(* IEC 61131-3 sources: generating_plc_code_with_llms/Code#1/ChatGPT_4/second run, 21 files *)

(* ---- 14.st ---- *)
// 60.33s
// 2
FUNCTION FC1001 : BOOL
VAR_INPUT
    measuredValue : REAL;  // Sensor reading
    switchingValue : REAL; // Predetermined switching value
    hysteresis : REAL;     // Hysteresis in percentage of the switching value
END_VAR

VAR
    hysteresisValue : REAL;
    static lastState : BOOL := FALSE;
END_VAR

// Calculate the hysteresis value
hysteresisValue := switchingValue * (hysteresis / 100.0);

// Switching logic with hysteresis
IF measuredValue > (switchingValue + hysteresisValue) THEN
    lastState := TRUE;  // Turn on the output
ELSIF measuredValue < (switchingValue - hysteresisValue) THEN
    lastState := FALSE; // Turn off the output
END_IF

FC1001 := lastState;

END_FUNCTION

(* ---- 15.st ---- *)
// 48.69s
// 2
FUNCTION FC1002 : BOOL
VAR_INPUT
    sensorDetected : BOOL; // TRUE if ultrasonic sensor detects something
    switchEA : BOOL;       // TRUE if the monitoring system is switched on
END_VAR

VAR_OUTPUT
    hornPHU : BOOL;        // Horn for acoustic warning signal
    alarmPAL : BOOL;       // Alarm signal
    indicatorP1 : BOOL;    // Indicator for monitoring system status
END_VAR

VAR
    detectionStartTime : TIME;
    systemActive : BOOL;
    static lastDetectionTime : TIME := 0;
END_VAR

// System control logic
IF switchEA THEN
    indicatorP1 := TRUE;  // Monitoring system is active
    systemActive := TRUE;

    IF sensorDetected THEN
        IF NOT hornPHU THEN
            detectionStartTime := TIME();  // Start the detection timer
        END_IF

        hornPHU := TRUE;  // Activate horn

        // Check if detection lasts longer than 3 seconds
        IF TIME() - detectionStartTime > T#3s THEN
            hornPHU := FALSE;   // Turn off horn
            alarmPAL := TRUE;   // Activate alarm
        END_IF
    ELSE
        hornPHU := FALSE;
        alarmPAL := FALSE;
        detectionStartTime := 0;
    END_IF
ELSE
    // Reset all outputs and states when the system is switched off
    hornPHU := FALSE;
    alarmPAL := FALSE;
    indicatorP1 := FALSE;
    systemActive := FALSE;
    detectionStartTime := 0;
END_IF

FC1002 := systemActive;

END_FUNCTION

(* ---- 18.st ---- *)
// 34.21s
// 4
FUNCTION FC1003 : REAL
VAR_INPUT
    digitalValue : REAL;   // Digital input value (e.g., 0 to 255)
    IN_MIN : REAL;         // Lower limit of the input range
    IN_MAX : REAL;         // Upper limit of the input range
    OUT_MIN : REAL;        // Lower limit of the output range (e.g., -20°C)
    OUT_MAX : REAL;        // Upper limit of the output range (e.g., 40°C)
END_VAR

VAR
    scaleFactor : REAL;
    offset : REAL;
END_VAR

BEGIN
    // Calculate the scale factor and offset for linear mapping
    scaleFactor := (OUT_MAX - OUT_MIN) / (IN_MAX - IN_MIN);
    offset := OUT_MIN - scaleFactor * IN_MIN;

    // Apply linear mapping
    FC1003 := scaleFactor * digitalValue + offset;
END_FUNCTION

(* ---- 19.st ---- *)
// 39.94s
// 2
FUNCTION_BLOCK FB1005
VAR_INPUT
    Laser1 : REAL;      // Measurement from Laser 1
    Laser2 : REAL;      // Measurement from Laser 2
    S1 : BOOL;          // Sensor to start/end measurement
    V_MAX : REAL;       // Upper tolerance limit
    V_MIN : REAL;       // Lower tolerance limit
END_VAR

VAR_OUTPUT
    M_MAX : REAL;       // Maximum measured thickness
    M_MIN : REAL;       // Minimum measured thickness
    P1 : BOOL;          // Reject indicator
END_VAR

VAR
    measuring : BOOL := FALSE;  // Indicates if currently measuring
    currentThickness : REAL;
END_VAR

BEGIN
    IF S1 THEN
        IF NOT measuring THEN
            // Start of a new measurement
            M_MAX := -REAL_MAX;
            M_MIN := REAL_MAX;
            measuring := TRUE;
            P1 := FALSE;
        END_IF

        // Calculate current thickness
        currentThickness := ABS(Laser1 - Laser2);

        // Update M_MAX and M_MIN
        IF currentThickness > M_MAX THEN
            M_MAX := currentThickness;
        END_IF

        IF currentThickness < M_MIN THEN
            M_MIN := currentThickness;
        END_IF

        // Check if the current measurement is out of tolerance
        IF (M_MAX > V_MAX) OR (M_MIN < V_MIN) THEN
            P1 := TRUE;  // Plate is scrap
        END_IF
    ELSE
        IF measuring THEN
            // End of measurement
            measuring := FALSE;
        END_IF
    END_IF
END_FUNCTION_BLOCK

(* ---- 21.st ---- *)
// 119.91s
// 3
FUNCTION_BLOCK BURNER
VAR_INPUT
    IN : BOOL;                // Start signal
    OVER_TEMP : BOOL;         // Boiler over-temperature signal
    OIL_TEMP : BOOL;          // Oil temperature readiness signal
    STAGE2 : BOOL;            // Signal to start stage 2
    RST : BOOL;               // Reset signal
END_VAR

VAR_OUTPUT
    PRE_HEAT : BOOL;          // Pre-heating signal
    MOTOR : BOOL;             // Motor operation signal
    IGNITION : BOOL;          // Ignition signal
    OIL_VALVE : BOOL;         // Oil valve open signal
    FAIL : BOOL;              // Failure signal
    STATUS : INT;             // Status code output
END_VAR

VAR
    TIMER : TON;              // Timer for managing delays
    currentStage : INT := 0;  // Current operation stage
    lockoutTimer : TON;       // Timer for managing lockout period
END_VAR

// Constants for timing (to be adjusted as per requirements)
VAR CONSTANT
    PRE_HEAT_TIME : TIME := T#30s;
    PRE_VENTILATION_TIME : TIME := T#15s;
    PRE_IGNITE_TIME : TIME := T#5s;
    SAFETY_TIME : TIME := T#10s;
    POST_IGNITE_TIME : TIME := T#5s;
    STAGE2_DELAY : TIME := T#60s;
    LOCKOUT_TIME : TIME := T#300s;
    MULTIPLE_IGNITION : BOOL := TRUE;  // Can be set based on requirements
END_VAR

// State machine logic
IF OVER_TEMP THEN
    // Immediate stop and report error 9
    STATUS := 9;
    FAIL := TRUE;
    ResetOutputs();
ELSIF RST AND NOT lockoutTimer.Q THEN
    // Resetting the burner
    FAIL := FALSE;
    STATUS := 110; // Standby
    currentStage := 0;
    ResetOutputs();
ELSIF IN THEN
    CASE currentStage OF
    0:  // Start sequence
        PRE_HEAT := TRUE;
        TIMER(IN := TRUE, PT := PRE_HEAT_TIME);
        IF OIL_TEMP THEN
            currentStage := 1;
            PRE_HEAT := FALSE;
            MOTOR := TRUE;
        ELSIF TIMER.Q THEN
            // Pre-heat failure
            FAIL := TRUE;
            STATUS := 1;
            currentStage := -1;  // Move to error state
        END_IF;
    1:  // Motor and ventilation
        TIMER(IN := TRUE, PT := PRE_VENTILATION_TIME);
        IF TIMER.Q THEN
            currentStage := 2;
            MOTOR := FALSE;  // Assuming motor should stop before ignition, adjust as needed
            IGNITION := TRUE;
        END_IF;
    2:  // Ignition and oil valve
        TIMER(IN := TRUE, PT := PRE_IGNITE_TIME);
        IF TIMER.Q THEN
            OIL_VALVE := TRUE;
            TIMER(IN := TRUE, PT := SAFETY_TIME);  // Start safety timer
            currentStage := 3;
        END_IF;
    3:  // Safety check
        IF NOT TIMER.Q THEN
            // Assume flame detected, proceed
            STATUS := 112;  // Burner running on stage 1
            currentStage := 4;
        ELSE
            // Safety time passed without flame
            FAIL := TRUE;
            STATUS := 4;
            currentStage := -1;  // Move to error state
        END_IF;
    4:  // Stage 2 check
        IF STAGE2 THEN
            TIMER(IN := TRUE, PT := STAGE2_DELAY);
            IF TIMER.Q THEN
                STATUS := 113;  // Burner running at stage 2
                // Implement stage 2 functionality as required
            END_IF;
        END_IF;
    -1: // Error state
        ResetOutputs();
        lockoutTimer(IN := TRUE, PT := LOCKOUT_TIME);  // Start lockout timer
        IF lockoutTimer.Q THEN
            // Lockout period finished, ready for reset
            currentStage := 0;
            FAIL := FALSE;
            STATUS := 110; // Back to standby after reset
        END_IF;
    END_CASE;
END_IF;

// Helper procedure to reset outputs
PROCEDURE ResetOutputs();
BEGIN
    PRE_HEAT := FALSE;
    MOTOR := FALSE;
    IGNITION := FALSE;
    OIL_VALVE := FALSE;
    TIMER(IN := FALSE, PT := T#0s);  // Reset timer
END_PROCEDURE

END_FUNCTION_BLOCK

(* ---- 1.st ---- *)
//16.57s
//4
PROGRAM AlarmControl
VAR
    xAlarm1: BOOL; // Alarm 1
    xAlarm2: BOOL; // Alarm 2
    xAllOn: BOOL;  // Signal to set all alarms
    xAllOff: BOOL; // Signal to reset all alarms
END_VAR

// When the xAllOn signal is active, set both alarms to TRUE
IF xAllOn THEN
    xAlarm1 := TRUE;
    xAlarm2 := TRUE;
    // Reset the signals after processing
    xAllOn := FALSE;
END_IF

// When the xAllOff signal is active, set both alarms to FALSE
IF xAllOff THEN
    xAlarm1 := FALSE;
    xAlarm2 := FALSE;
    // Reset the signals after processing
    xAllOff := FALSE;
END_IF

END_PROGRAM

(* ---- 10.st ---- *)
//16.26s
//4
PROGRAM SigmoidFunction
VAR
    x: REAL;        // Input for the sigmoid function
    sigmoid: REAL;  // Result of the sigmoid function
END_VAR

// Calculate the sigmoid function
sigmoid := 1 / (1 + EXP(-x));

END_PROGRAM

(* ---- 11.st ---- *)
//19.66s
//4
PROGRAM SignFunction
VAR
    x: REAL;        // Input variable
    signum: INT;    // Output variable (-1, 0, 1)
END_VAR

// Calculate the signum of the variable x
IF x < 0 THEN
    signum := -1;
ELSIF x > 0 THEN
    signum := 1;
ELSE
    signum := 0;
END_IF;

END_PROGRAM

(* ---- 12.st ---- *)
//14.62s
//4
PROGRAM HyperbolicSine
VAR
    x: REAL;           // Input variable
    sinh_x: REAL;      // Result of hyperbolic sine of x
END_VAR

// Calculate the hyperbolic sine of x
sinh_x := (EXP(x) - EXP(-x)) / 2;

END_PROGRAM

(* ---- 13.st ---- *)
//30.69s
//2
PROGRAM SearchNumber
VAR
    RandomNumbers: ARRAY[1..100] OF INT; // Array containing 100 random numbers
    Found: BOOL; // TRUE if the number 10 is found, FALSE otherwise
    i: INT; // Index used for iterating through the list
END_VAR

i := 1; // Initialize index
Found := FALSE; // Initialize Found as FALSE

REPEAT
    IF RandomNumbers[i] = 10 THEN
        Found := TRUE; // Set Found to TRUE if number 10 is found
        EXIT; // Exit the loop if number 10 is found
    END_IF;
    i := i + 1; // Increment index
UNTIL i > 100; // Continue until the end of the list is reached

IF Found THEN
    // Number 10 was found in the list
    // Additional actions can be taken here if necessary
ELSE
    // Number 10 was not found in the list
    // Additional actions can be taken here if necessary
END_IF;

END_PROGRAM

(* ---- 16.st ---- *)
//41.0s
//4
PROGRAM TrafficLightControl
VAR
    North_green, North_yellow, North_red: BOOL; // North traffic lights
    East_green, East_yellow, East_red: BOOL; // East traffic lights
    CycleTimer: TON; // Timer for controlling the cycle
END_VAR

// Start the cycle timer
CycleTimer(IN:=TRUE, PT:=T#10000ms);

// Control North traffic light
IF CycleTimer.ET < T#5000ms THEN
    // Between 0ms and 5000ms, North is green and East is red
    North_green := TRUE;
    North_yellow := FALSE;
    North_red := FALSE;

    East_green := FALSE;
    East_yellow := FALSE;
    East_red := TRUE;
ELSIF CycleTimer.ET < T#5500ms THEN
    // Between 5000ms and 5500ms, North turns yellow
    North_green := FALSE;
    North_yellow := TRUE;
    North_red := FALSE;

    East_green := FALSE;
    East_yellow := FALSE;
    East_red := TRUE;
ELSE
    // After 5500ms, North is red
    North_green := FALSE;
    North_yellow := FALSE;
    North_red := TRUE;
END_IF;

// Control East traffic light
IF CycleTimer.ET >= T#5500ms AND CycleTimer.ET < T#9500ms THEN
    // Between 5500ms and 9500ms, East is green
    East_green := TRUE;
    East_yellow := FALSE;
    East_red := FALSE;
ELSIF CycleTimer.ET >= T#9500ms THEN
    // Between 9500ms and 10000ms, East turns yellow
    East_green := FALSE;
    East_yellow := TRUE;
    East_red := FALSE;
END_IF;

// Reset the timer after the cycle completes
IF CycleTimer.ET >= CycleTimer.PT THEN
    CycleTimer.IN := FALSE; // Stop the timer
    CycleTimer( IN:=FALSE ); // Reset the timer
    CycleTimer.IN := TRUE; // Restart the timer for the next cycle
END_IF;

END_PROGRAM

(* ---- 17.st ---- *)
//39.92s
//2
PROGRAM WeatherStation
VAR
    aiTemperature: INT; // Analog input value for temperature
    aiHumidity: INT; // Analog input value for humidity
    rTemperatureC: REAL; // Scaled temperature in degrees Celsius
    rHumidityPct: REAL; // Scaled humidity in percent
    DisplayText: STRING; // Text to be displayed
END_VAR

// Assuming aiTemperature and aiHumidity are scaled appropriately to 0-100% for the 0-32767 range
rTemperatureC := (REAL(aiTemperature) / 32767) * 100; // Convert to degrees Celsius (example scaling)
rHumidityPct := (REAL(aiHumidity) / 32767) * 100; // Convert to percent (example scaling)

IF rTemperatureC < 18 THEN
    DisplayText := 'Cold';
ELSIF rTemperatureC > 25 THEN
    DisplayText := 'Hot';
ELSE
    // Temperature is between 18 and 25 degrees Celsius, check humidity
    IF rHumidityPct >= 40 AND rHumidityPct <= 75 THEN
        DisplayText := 'Opt'; // Optimum conditions
    ELSE
        DisplayText := 'Temp. OK'; // Temperature is okay, but humidity is not in the optimum range
    END_IF;
END_IF;

END_PROGRAM

(* ---- 2.st ---- *)
//18.14s
//4
FUNCTION Factorial: LINT
VAR_INPUT
    n: INT; // Input value to calculate the factorial of
END_VAR
VAR
    i: INT;
    result: LINT := 1; // Initialize result to 1 (0! = 1)
END_VAR

FOR i := 1 TO n DO
    result := result * i;
END_FOR

Factorial := result; // Return the factorial result
END_FUNCTION

PROGRAM BinomialCoefficient
VAR
    n: INT; // Total number of items
    k: INT; // Number of items to choose
    binomCoeff: LINT; // Binomial coefficient result
END_VAR

// Ensure that 0 <= k <= n, otherwise the binomial coefficient is not defined
IF k >= 0 AND k <= n THEN
    binomCoeff := Factorial(n) / (Factorial(k) * Factorial(n - k));
ELSE
    binomCoeff := 0; // If the condition is not met, the result is 0
END_IF

END_PROGRAM

(* ---- 20.st ---- *)
// 48.24s
// 4
PROGRAM InterlockProgram
VAR
    I1, I2 : BOOL;       // Inputs
    Q1, Q2 : BOOL;       // Outputs
    TL : TIME;           // Dead time between outputs
    LastQ1Time, LastQ2Time : TIME;  // Time trackers for Q1 and Q2
END_VAR

BEGIN
    // Update time trackers
    IF Q1 THEN
        LastQ1Time := TIME();
    END_IF
    IF Q2 THEN
        LastQ2Time := TIME();
    END_IF

    // Logic for Q1
    IF I1 AND NOT Q2 AND (TIME() - LastQ2Time > TL) THEN
        Q1 := TRUE;
    ELSE
        Q1 := FALSE;
    END_IF

    // Logic for Q2
    IF I2 AND NOT Q1 AND (TIME() - LastQ1Time > TL) THEN
        Q2 := TRUE;
    ELSE
        Q2 := FALSE;
    END_IF
END_PROGRAM

(* ---- 3.st ---- *)
//24.56s
//2
FUNCTION Fibonacci: LINT
VAR_INPUT
    n: INT; // The n-th Fibonacci number to calculate
END_VAR
VAR
    a: LINT := 0; // First number in the sequence
    b: LINT := 1; // Second number in the sequence
    i: INT;
    temp: LINT;
END_VAR

IF n = 0 THEN
    RETURN 0; // The 0th Fibonacci number is 0
ELSIF n = 1 THEN
    RETURN 1; // The 1st Fibonacci number is 1
ELSE
    FOR i := 2 TO n DO
        temp := a + b; // Calculate the next Fibonacci number
        a := b; // Move to the next number in the sequence
        b := temp; // Set the new value
    END_FOR
    RETURN b; // The n-th Fibonacci number
END_IF
END_FUNCTION

PROGRAM Main
VAR
    n: INT := 10; // Example: Calculate the 10th Fibonacci number
    fibNumber: LINT; // Variable to store the result
END_VAR

fibNumber := Fibonacci(n); // Call the function and store the result

END_PROGRAM

(* ---- 4.st ---- *)
//38.21s
//2
PROGRAM FillLevelCheck
VAR
    nAnalogValue: INT; // Raw analog value from the sensor (0 - 32767)
    rFillLevel: REAL;  // Scaled fill level (0.0 - 100.0%)
    xLowLevel: BOOL;   // Output for low level
    xOkLevel: BOOL;    // Output for ok level
    xHighLevel: BOOL;  // Output for high level
    xWarningHorn: BOOL; // Output for warning horn (< 1% level)
END_VAR

// Scale the analog value to a percentage (0-100%)
rFillLevel := (REAL(nAnalogValue) / 32767) * 100;

// Determine the range of the fill level and set outputs accordingly
CASE TRUE OF
    rFillLevel < 1.0:
        xWarningHorn := TRUE; // Activate the warning horn
        xLowLevel := FALSE;
        xOkLevel := FALSE;
        xHighLevel := FALSE;
    rFillLevel >= 1.0 AND rFillLevel < 20.0:
        xLowLevel := TRUE;
        xOkLevel := FALSE;
        xHighLevel := FALSE;
        xWarningHorn := FALSE; // Deactivate the warning horn
    rFillLevel >= 20.0 AND rFillLevel <= 80.0:
        xLowLevel := FALSE;
        xOkLevel := TRUE;
        xHighLevel := FALSE;
        xWarningHorn := FALSE; // Deactivate the warning horn
    rFillLevel > 80.0:
        xLowLevel := FALSE;
        xOkLevel := FALSE;
        xHighLevel := TRUE;
        xWarningHorn := FALSE; // Deactivate the warning horn
    ELSE
        xLowLevel := FALSE;
        xOkLevel := FALSE;
        xHighLevel := FALSE;
        xWarningHorn := FALSE; // Default case, no level detected
END_CASE

END_PROGRAM

(* ---- 5.st ---- *)
//44.26s
//2
PROGRAM GateController
VAR
    Start_Loop: BOOL; // Control variable to start the timer loop
    One_Hour_Timer: TON; // Timer that counts up to 1 hour
    Gate_Open: BOOL; // Indicates if the gate is open
    Sense_App: BOOL; // Senses the app signal
    Sense_Car: BOOL; // Senses the car signal
    Auth_String: STRING; // Received authorization string
    CONST my_defined_str: STRING := 'YourAuthString'; // Replace with your actual auth string
END_VAR

// Start the one hour timer when Start_Loop is FALSE
IF NOT Start_Loop THEN
    One_Hour_Timer(IN := TRUE, PT := T#1h); // Set the preset time to 1 hour
ELSE
    One_Hour_Timer(IN := FALSE, PT := T#1h);
END_IF

// Check for timeout to close the gate
IF One_Hour_Timer.Q AND Gate_Open THEN
    Gate_Open := FALSE; // Close the gate
END_IF

// Check for app or car sense and correct authorization string
IF (Sense_App OR Sense_Car) AND (Auth_String = my_defined_str) THEN
    Gate_Open := TRUE; // Open the gate
END_IF

// Reset the timer if the gate is manually closed
IF NOT Gate_Open THEN
    One_Hour_Timer(IN := FALSE); // Reset the timer
    Start_Loop := TRUE; // Ready to start the loop again
END_IF

END_PROGRAM

(* ---- 6.st ---- *)
//49.85s
// 4
PROGRAM CraneLift
VAR
    // Conveyor belts
    doConvTop: BOOL;    // Actuator for the top conveyor belt
    doConvBottom: BOOL; // Actuator for the bottom conveyor belt
    doConvLift: BOOL;   // Actuator for the lift conveyor belt
    // Light barriers
    diConvTop: BOOL;    // Sensor for the top conveyor belt
    diConvBottom: BOOL; // Sensor for the bottom conveyor belt
    // Lift positions
    doLiftTop: BOOL;    // Move lift to the top position
    doLiftBottom: BOOL; // Move lift to the bottom position
    doLiftUnload: BOOL; // Move lift to the unloading position
    // Lift position sensors
    diLiftTop: BOOL;    // Sensor for the lift at the top position
    diLiftBottom: BOOL; // Sensor for the lift at the bottom position
    diLiftUnload: BOOL; // Sensor for the lift at the unloading position
    // Box sensors
    diBoxLift: BOOL;    // Sensor for the box at the lift
    // Control flags
    bRequestTop: BOOL;    // Flag indicating a request for the top position
    bRequestBottom: BOOL; // Flag indicating a request for the bottom position
    bUnloadProcess: BOOL; // Flag indicating the lift is in the unloading process
END_VAR

// Logic for detecting crates and requesting lift
IF diConvTop THEN
    doConvTop := FALSE; // Stop the top conveyor belt
    bRequestTop := TRUE; // Set the request flag for top position
END_IF

IF diConvBottom THEN
    doConvBottom := FALSE; // Stop the bottom conveyor belt
    bRequestBottom := TRUE; // Set the request flag for bottom position
END_IF

// Logic for moving lift to requested position
IF bRequestTop AND NOT bRequestBottom AND NOT diLiftTop THEN
    doLiftTop := TRUE; // Request lift to move to top position
    doLiftBottom := FALSE; // Ensure lift is not moving to bottom
    doLiftUnload := FALSE; // Ensure lift is not moving to unload
ELSIF bRequestBottom AND NOT bRequestTop AND NOT diLiftBottom THEN
    doLiftBottom := TRUE; // Request lift to move to bottom position
    doLiftTop := FALSE; // Ensure lift is not moving to top
    doLiftUnload := FALSE; // Ensure lift is not moving to unload
END_IF

// Logic for operating lift conveyor belt
IF (diLiftTop AND bRequestTop) OR (diLiftBottom AND bRequestBottom) THEN
    doConvLift := TRUE; // Turn on the lift conveyor belt
    // Reset request flags as the lift is now servicing the request
    bRequestTop := FALSE;
    bRequestBottom := FALSE;
    bUnloadProcess := TRUE; // Start the unloading process
ELSE
    doConvLift := FALSE; // Turn off the lift conveyor belt
END_IF

// Logic for box on lift conveyor belt
IF diBoxLift AND bUnloadProcess THEN
    // Box is completely at the lift, move to unloading position
    doLiftUnload := TRUE;
    // Turn off lift conveyor belt as box is now moving to unload
    doConvLift := FALSE;
END_IF

// Logic for unloading box
IF diLiftUnload AND bUnloadProcess THEN
    // Box has reached unloading position, conveyor belt unloads the box
    doConvLift := TRUE;
    // Once the box has left the lift, it is free for the next request
    IF NOT diBoxLift THEN
        bUnloadProcess := FALSE;
        doLiftUnload := FALSE;
    END_IF
END_IF

END_PROGRAM

(* ---- 7.st ---- *)
//31.16s
// 4
PROGRAM CraneLoadCalculation
VAR
    aiLoadReceptor1: INT; // Analog input from load receptor 1
    aiLoadReceptor2: INT; // Analog input from load receptor 2
    aiLoadReceptor3: INT; // Analog input from load receptor 3
    aiLoadReceptor4: INT; // Analog input from load receptor 4
    aiLoadReceptor5: INT; // Analog input from load receptor 5
    rTotalLoad: REAL;     // Variable for total load
    rAverageLoad: REAL;   // Variable for average load
END_VAR

VAR CONSTANT
    NUM_RECEPTORS: INT := 5; // Constant for the number of load receptors
    MAX_ANALOG_VALUE: INT := 32767; // Constant for maximum analog value
END_VAR

VAR
    arLoadValues: ARRAY[1..NUM_RECEPTORS] OF INT; // Array to store load values
    i: INT; // Loop counter
END_VAR

// Assign analog values to the array
arLoadValues[1] := aiLoadReceptor1;
arLoadValues[2] := aiLoadReceptor2;
arLoadValues[3] := aiLoadReceptor3;
arLoadValues[4] := aiLoadReceptor4;
arLoadValues[5] := aiLoadReceptor5;

rTotalLoad := 0; // Initialize total load

// Calculate total load using a FOR loop
FOR i := 1 TO NUM_RECEPTORS DO
    rTotalLoad := rTotalLoad + arLoadValues[i];
END_FOR

// Calculate average load
rAverageLoad := rTotalLoad / NUM_RECEPTORS;

END_PROGRAM

(* ---- 8.st ---- *)
//36.73s
//2
PROGRAM LambertWFunction
VAR
    x: REAL; // The input value for which you want to find the Lambert W
    w: REAL; // The approximation of the Lambert W function result
    w_prev: REAL; // The previous approximation of W to check for convergence
    e_to_w: REAL; // e raised to the power of the current approximation of W
    tolerance: REAL := 1e-5; // Tolerance for the approximation
    max_iterations: INT := 100; // Maximum number of iterations
    iteration: INT; // Current iteration counter
END_VAR

// Initial guess, works well for small x values
IF x < 1 THEN
    w := x;
ELSE
    w := LOG(x); // Natural logarithm of x as the initial guess for larger values
END_IF

iteration := 0;
REPEAT
    iteration := iteration + 1;
    e_to_w := EXP(w); // e raised to the current approximation of W
    w_prev := w;
    // Halley's method for next approximation
    w := w - ((w * e_to_w - x) / (e_to_w * (w + 1) - ((w + 2) * (w * e_to_w - x) / (2 * w + 2))));
UNTIL (ABS(w - w_prev) <= tolerance) OR (iteration >= max_iterations);

// The result is in w
END_PROGRAM

(* ---- 9.st ---- *)
//22.72s
//4
PROGRAM LeapYearCheck
VAR
    YEAR: INT; // The year to check
    IsLeapYear: BOOL; // Output: TRUE if 'YEAR' is a leap year, otherwise FALSE
END_VAR

// Check if the year is a leap year
IsLeapYear := FALSE; // Initialize as FALSE

IF (YEAR MOD 4 = 0) THEN
    IF (YEAR MOD 100 = 0) THEN
        IF (YEAR MOD 400 = 0) THEN
            IsLeapYear := TRUE; // Year is divisible by 400, it's a leap year
        END_IF;
    ELSE
        IsLeapYear := TRUE; // Year is not a century and is divisible by 4, it's a leap year
    END_IF;
END_IF;

END_PROGRAM
